{attribute 'GeneratedUsingTerminal: EL7031-0000-0016'}
{attribute addProperty BoxType "EL7031-0000-0016"}
{attribute addProperty Id "VelocityAT %Q*INT2"}
{attribute addProperty CRC "2759475009"}
{attribute addProperty Size "2"}
TYPE STM_Velocity_A47A3F41 :
STRUCT
	{attribute addProperty Name "Velocity"}
	Velocity AT %Q* : INT;
END_STRUCT
END_TYPE

(* stored: Version 1.2.0.0, ProductVersion 3.1.4024.9
   DUT STM_Velocity_A47A3F41: Id {e157cef5-cfe7-4d8b-b0fd-d2372e542c76} *)
